Staubli VAL3: getPoint.pgx

public program getPoint(point& x_pPoint[], bool x_bCycle, num x_nIndex)
begin
end
